Staubli VAL3: showStatus.pgx

program showStatus()
  local joint l_jHere
  local point l_pHere
  local string l_sMessage[2]
  local tool l_tTool
  local num l_nIndexTool
  local frame l_fFrame
begin
  //
  // show an dialog box with
  // the current Joint/cartesian position
  //
  l_fFrame=world
  l_fFrame.trsf=saveData:fFrameItem[saveData:nFrameActive].fFrame.trsf
  call trajType:getTool(l_nIndexTool)
  call tcp:getTool(l_tTool,l_nIndexTool)
  if cycleStatus:nWorkingStatus>1 and cycleStatus:nWorkingStatus<5 and cycleStatus:nWorkingMode==1
    // set a timer of x second then the message disappear ..
    if !bTrigger
      nClockStatus=clock()
      bTrigger=true
      bShowStatus=true
    endIf
    if clock()-nClockStatus<saveData:nTimeDialog
      if cycleStatus:nWorkingStatus==2
        l_jHere=herej()
        l_sMessage="J1:"+toString("7.1",l_jHere.j1)
        l_sMessage=l_sMessage+"  J2:"+toString("7.1",l_jHere.j2)
        l_sMessage=l_sMessage+"  J3:"+toString("7.1",l_jHere.j3)+"#"
        l_sMessage=l_sMessage+"J4:"+toString("7.1",l_jHere.j4)
        l_sMessage=l_sMessage+"  J5:"+toString("7.1",l_jHere.j5)
        l_sMessage=l_sMessage+"  J6:"+toString("7.1",l_jHere.j6)
      else
        l_pHere=here(l_tTool,l_fFrame)
        l_sMessage="X :"+toString("7.1",l_pHere.trsf.x)
        l_sMessage=l_sMessage+"  Y :"+toString("7.1",l_pHere.trsf.y)
        l_sMessage=l_sMessage+"  Z :"+toString("7.1",l_pHere.trsf.z)+"#"
        l_sMessage=l_sMessage+"RX:"+toString("7.1",l_pHere.trsf.rx)
        l_sMessage=l_sMessage+"  RY:"+toString("7.1",l_pHere.trsf.ry)
        l_sMessage=l_sMessage+"  RZ:"+toString("7.1",l_pHere.trsf.rz)
      endIf
      call use:timerDialog(l_sMessage,0)
    else
      // disable it
      bShowStatus=false
    endIf
  else
    // reset it
    if bTrigger and !cycleStatus:bCycle
      resetMotion()
    endIf
    bTrigger=false
    bShowStatus=false
  endIf
end
